(* IEC 61131-3 sources: NachHouse_CORE/V21/APP, 10 files *)

(* ---- _Nh_CFG.st ---- *)
VAR_GLOBAL
//	yVer	AT mRam[20000]	: NH_DBX_VER;            // verzia sa umiestni dalej do virtualne pamati. Na zaciatku sa pouzije a potom sa prepisuje datami
//   aDbx	AT mRam[0]	: NH_DBX;
   aCfg 	AT mRam[_Cfg0]	: ARRAY[1.._Nh_CFG] OF NH_CFG_CFG :=  [
			(cfg:='ROM',
                     ver:=1,
                     Siz   := SIZEOF(NH_ROM),                         // 1
                     al    := SIZEOF(NH_ROM.AL),
                     cx    := SIZEOF(NH_ROM.CX),
                     hw    := 0,                         // 1
                     io    := SIZEOF(NH_ROM.IO),                         // 1
                     me    := SIZEOF(NH_ROM.ME),                         // 1
                     cat   := 0,
                     fBr   := 14,
                     fSc   := 204,
                     mWsb  := 1,
                     mnu   := 25,
//                     wh    := 100,        // zobrazenie teploty v browse
                     ar2   := 1,
                     stp   := 0,

                     ref   := 252,
							del   := 1,
                     imp   := 1,
							bck	:= 1,
							RomIsZone:=1,

							NbrPoi:=1,
							),
         (cfg:='CAT',
                     ver:=0,
//                     Siz   := SIZEOF(NH_CAT),                         // 1
//                     al    := SIZEOF(NH_CAT.AL),
                     Siz   := 0,                         // 1
                     al    := 0,
                     cx    := 0,
                     hw    := 0,                         // 1
                     me    := 0,                         // 1
                     cat   := 0,
                     ar2   := 1,
                     stp   := 0,
                     fBr   := 12,
                     del   := 0,
                     ref   := 251,
							del   := 0,
                     imp   := 0,
							bck	:= 0,
                     ),

				(cfg:='ZON',
                     ver:=1,
                     Siz   := SIZEOF(NH_ROM),                         // 1
                     al    := SIZEOF(NH_ROM.AL),
                     cx    := SIZEOF(NH_ROM.CX),
                     hw    := 0,                         // 1
                     io    := SIZEOF(NH_ROM.IO),                         // 1
                     me    := SIZEOF(NH_ROM.ME),                         // 1
                     par   := 5,
                     fBr   := 14,
                     fSc   := 204,
                     mWsb  := 3,
                     mnu   := 24,
                     cat   := 0,
                     ar2   := 1,
                     stp   := 0,

                     ref   := 252,
							tgrp	:= 3,
							del   := 1,
                     imp   := 0,
							bck	:= 1,
							RomIsZone:=1,
			            ),
			(cfg:='SCN',                                                   // 4
                     ver:=1,
                     Siz   := SIZEOF(NH_SCN),
                     al    := SIZEOF(NH_SCN.AL),
                     cx    := SIZEOF(NH_SCN.CX),
                     me    := SIZEOF(NH_SCN.ME),
                     hw    := 0,                         // 1
							cat	:= 53,
                     sld   := 0,
                     par   := 10,
                     ou    := 1,
                     lst   := 1,
                     stp   := 1,
                     del   := 1,

                     fBr   := 5,
                     fSc   := 204,
                     mWsb  := 4,
                     mnu   := 93,
//                     analog:= 0,
                     tgrp  := 4,
//							analog:=true,
							zone	:=true,
							del   := 1,
                     imp   := 0,
							bck	:= 1,
							Visible:=1,
					      ),
			(cfg:='ACT',                                                   // 5
                     ver:=1,
                     Siz   := SIZEOF(NH_ACT),
                     al    := SIZEOF(NH_ACT.AL),
                     cx    := 0,
                     fBr   := 5,
                     fSc   := 204,
                     par   := 0,
                     cat   := 0,
							mWsb	:= 5,
                     mnu   := 94,
                     lst   := 1,
                     stp   := 1,
                     ou    := 0,
                     analog:= 0,
                     tgrp  := 5,
							zone	:=true,
							del   := 1,
                     imp   := 0,
							bck	:= 1,
							RomIsZone:=1,
							Visible:=1,
			            ),

         (cfg:='HET',                            		                    // 6
                     ver:=1,
                     Siz   := SIZEOF(NH_HET),
                     al    := SIZEOF(NH_HET.AL),
                     cx    := SIZEOF(NH_HET.CX),
                     hw    := 0,
                     me    := SIZEOF(NH_HET.ME),
                     io    := SIZEOF(NH_HET.IO),
                     fBR   := 23,
                     fSc   := 204,
                     mnu   := 28,
                     par   := 9,
          				mWsb	:= 6,
			            cat   := 5,
//                     cou   := 2,
                     sld   := 0,
//                     wh    := 100,        // zobrazenie teploty v browse
                     ou    := 0,       // ???? 23.11.2021
                     ref   := 251,
                     tgrp  := 6,
                    	lst	:= 1,
							del   := 1,
                     imp   := 0,
							bck	:= 1,
							ShwSta:=true,

							NbrPoi:=2,
							Imp_AL:=1,
                     ),

			(cfg:='KOT',                            	                       // 7
                     ver:=1,
                     Siz   := SIZEOF(NH_TVE),
                     al    := SIZEOF(NH_TVE.AL),
                     cx    := SIZEOF(NH_TVE.CX),
                     hw    := SIZEOF(NH_TVE.HW),
                     io    := SIZEOF(NH_TVE.IO),
                     me    := SIZEOF(NH_TVE.ME),
                     fBR   := 22,
                     mnu   := 36,
                     fSc   := 204,
                     cat   := 39,
                     sld   := 0,
                     par   := 0,
                     ou    := 1,
							del   := 0,
                     imp   := 1,
							bck	:= 1,
							Imp_AL:=1,
                     ),

			(cfg:='TVE',                            	                       // 8
                     ver:=1,
                     Siz   := SIZEOF(NH_TVE),
                     al    := SIZEOF(NH_TVE.AL),
                     cx    := SIZEOF(NH_TVE.CX),
                     hw    := SIZEOF(NH_TVE.HW),
                     io    := SIZEOF(NH_TVE.IO),
                     me    := SIZEOF(NH_TVE.ME),
                     fBR   := 22,
                     mnu   := 36,
                     fSc   := 204,
                     cat   := 39,
                     sld   := 0,
                     par   := 0,
                     ou    := 1,
							del   := 0,
                     imp   := 1,
							bck	:= 1,
							Imp_AL:=1,

                     ),
			(cfg:='CER',                               							  // 9
                     ver:=1,
                     Siz   := SIZEOF(NH_TVE),
                     al    := SIZEOF(NH_TVE.AL),
                     cx    := SIZEOF(NH_TVE.CX),
                     hw    := SIZEOF(NH_TVE.HW),
                     io    := SIZEOF(NH_TVE.IO),
                     me    := SIZEOF(NH_TVE.ME),
                     fBR   := 22,
                     mnu   := 36,
                     fSc   := 204,
                     cat   := 39,
                     sld   := 0,
                     par   := 0,
                     ou    := 1,
							del   := 0,
                     imp   := 1,
							bck	:= 1,
							Imp_AL:=1,

			            ),
         (cfg:='SVD',                                                      // 10
                     ver:=1,
                     Siz   := SIZEOF(NH_SVD),
                     al    := SIZEOF(NH_SVD.AL),
                     cx    := SIZEOF(NH_SVD.CX),
                     hw    := SIZEOF(NH_SVD.HW),
                     cat   := 1,
                     sld   := 0,
							lst	:= 1,
                     par   := 1,
                     ou    := 1,
                     fBr   := 43,
                     fSc   := 204,
                     mnu   := 45,
                     mWsb  := 10,
							ShwSta:=true,
                     del   := 0,
                     imp   := 1,
							bck	:= 1,
//                     adObr2:= 1,
			            ),
			(cfg:='SVA',                                                      // 11
                     ver:=1,
                     Siz   := SIZEOF(NH_SVA),
                     al    := SIZEOF(NH_SVA.AL),
                     cx    := SIZEOF(NH_SVA.CX),
                     hw    := SIZEOF(NH_SVA.HW),
                     cat   := 1,
							lst	:= 1,
                     sld   := 1,
                     par   := 2,
                     ou    := 1,
                     fBr   := 43,
                     fSc   := 204,
                     mWsb  := 11,
                     mnu   := 45,
                     analog:=true,
							ShwSta:=true,
                     del   := 0,
                     imp   := 1,
							bck	:= 1,
			            ),
			(cfg:='RGB',                                                      // 12
                     ver:=1,
                     Siz   := SIZEOF(NH_RGB),
                     al    := SIZEOF(NH_RGB.AL),
                     cx    := SIZEOF(NH_RGB.CX),
                     hw    := SIZEOF(NH_RGB.HW),
                     cat   := 1,
                     sld   := 1,
							lst	:= 1,
                     par   := 3,
                     ou    := 1,
                     fBr   := 43,
                     fSc   := 204,
                     mWsb  := 11,
                     mnu   := 46,
                     analog:=true,
                     del   := 0,
                     imp   := 1,
							bck	:= 1,
                     ),
			(cfg:='WSB',                                                      // 13
                     ver:=1,
                     Siz   := SIZEOF(NH_WSB),
                     al    := SIZEOF(NH_WSB.AL),
                     cx    := SIZEOF(NH_WSB.CX),
                     hw    := SIZEOF(NH_WSB.HW),
                     me    := SIZEOF(NH_WSB.ME),
                     fSc   := 204,
                     mnu   := 27,
                     cat   := 24,
                     sld   := 0,
                     par   := 4,
                     ref   := 252,
                     body  := 1,
                     tgrp  := 13,
                     del   := 0,
                     imp   := 1,
							bck	:= 1,
							led	:= 1,
                     ),
			(cfg:='TLA',                                       			     // 14

                     ver:=1,
                     Siz   := SIZEOF(NH_TLA),
                     al    := SIZEOF(NH_TLA.AL),
                     cx    := SIZEOF(NH_TLA.CX),
                     hw    := SIZEOF(NH_TLA.HW),
                     me    := SIZEOF(NH_TLA.ME),
                     fSc   := 204,
                     mnu   := 27,

//                     iov   := 1,
                     cat   := 24,
                     sld   := 0,
                     par   := 4,
                     ref   := 252,
                     body  := 1,
                     tgrp  := 13,
                     del   := 0,
                     imp   := 1,
							bck	:= 1,
                     ),
   	   (cfg:='PIR',                                                     // 15
                     ver:=1,
                     Siz   := SIZEOF(NH_PIR),
                     al    := SIZEOF(NH_PIR.AL),
                     cx    := SIZEOF(NH_PIR.CX),
                     hw    := SIZEOF(NH_PIR.HW),
                     me    := 0,	//SIZEOF(NH_PIR.ME),
                     cat   := 15,
                     fBr   := 15,
                     fSc   := 204,
                     mWsb  := 15,
                     mnu   := 56,
                     par   := 7,
                     body  := 1,
                     tgrp  := 15,
                     del   := 0,
                     imp   := 1,
							bck	:= 1,
                     ),

			(cfg:='TER',                                                      // 16
                     ver:=1,
                     Siz   := SIZEOF(NH_TER),
                     al    := SIZEOF(NH_TER.AL),
                     cx    := SIZEOF(NH_TER.CX),
                     hw    := SIZEOF(NH_TER.HW),
                     me    := SIZEOF(NH_TER.ME),
                     cat   := 14,
//                     wh    := 100,        // zobrazenie teploty v browse
                     par   := 0,
                     fBr   := 20,
                     fSc   := 204,
                     mnu   := 34,
                     tgrp  := 16,
							//   iov	:= 100,
							ShwSta:=false,
							analog:=true,
							zone	:=true,
                     del   := 1,
                     imp   := 1,
							bck	:= 1,
                     ),

			(cfg:='TEH',                                                      // 17
                     ver:=1,
                     Siz   := SIZEOF(NH_TER),
                     al    := SIZEOF(NH_TER.AL),
                     cx    := SIZEOF(NH_TER.CX),
                     hw    := SIZEOF(NH_TER.HW),
                     me    := SIZEOF(NH_TER.ME),
//                     wh    := 100,        // zobrazenie teploty v browse
                     cat   := 39,
                     par   := 0,
                     fBr   := 20,
                     fSc   := 204,
                     mnu   := 34,
                     tgrp  := 16,
                     //iov   := 100,
							analog:=true,
                     del   := 1,
                     imp   := 1,
							bck	:= 1,
                     ),
			(cfg:='TEK',                                                      // 18
                     ver:=1,
                     Siz   := SIZEOF(NH_TER),
                     al    := SIZEOF(NH_TER.AL),
                     cx    := SIZEOF(NH_TER.CX),
                     hw    := SIZEOF(NH_TER.HW),
                     me    := SIZEOF(NH_TER.ME),
//                     wh    := 100,        // zobrazenie teploty v browse
                     cat   := 39,
                     par   := 0,
                     fBr   := 20,
                     fSc   := 204,
                     mnu   := 34,
							analog:=true,
                     tgrp  := 16,
                     //  iov   := 100,
                     del   := 1,
                     imp   := 1,
							bck	:= 1,
                     ),
			(cfg:='LUX',                                                      // 19
                     ver:=1,
                     Siz   := SIZEOF(NH_LUX),
                     al    := SIZEOF(NH_LUX.AL),
                     cx    := SIZEOF(NH_LUX.CX),
                     hw    := SIZEOF(NH_LUX.HW),
                     me    := SIZEOF(NH_LUX.ME),
//                     wh    := 101,        // zobrazenie % v browse
                     cat   := 16,
                     par   := 0,
                     fBr   := 20,

                     fSc   := 204,
                     mnu   := 59,

                     tgrp  := 16,
                     //  iov   := 101,
							analog:=true,
							zone	:=true,
                     del   := 0,
                     imp   := 1,
							bck	:= 1,
                     ),
                                                                           // 20
	      (cfg:='FAV',
                     ver:=1,
                     Siz   := SIZEOF(NH_FAV),
                     al    := 0,
                     cx    := SIZEOF(NH_FAV.CX),
                     fav   := 0,
                     par   := 0,

                     del   := 1,
                     imp   := 0,
							bck	:= 0,
                     ),

	      (cfg:='ZAS',                                                        // 21
                     ver:=1,
                     Siz   := SIZEOF(NH_SVD),
                     al    := SIZEOF(NH_SVD.AL),
                     cx    := SIZEOF(NH_SVD.CX),
                     hw    := SIZEOF(NH_SVD.HW),
                     cat   := 2,
							lst	:= 1,
                     par   := 1,
                     sld   := 0,
                     ou    := 1,
                     fBr   := 43,
                     fSc   := 204,
                     mnu   := 45,
                     mWsb  := 10,
                     del   := 0,
                     imp   := 1,
							bck	:= 1,

//                     adObr2:= 1,
                     ),

			(cfg:='USR',
                     ver:=1,
                     Siz   := SIZEOF(NH_USR),  					              // 22  uzivatelia
                     al    := 0,
                     cx    := SIZEOF(NH_USR.CX),
                     stp   := 0,
                     cat   := 31,
                     par   := 0,
                     ref   := 254,

                     del   := 1,
                     imp   := 0,
							bck	:= 1,
                     ),
			(cfg:='VEN',                                                      // 23 TVE pre Vetranie // ako TVE pre HET
                     ver:=1,
                     Siz   := SIZEOF(NH_TVE),
                     al    := SIZEOF(NH_TVE.AL),
                     cx    := SIZEOF(NH_TVE.CX),
                     hw    := SIZEOF(NH_TVE.HW),
                     io    := SIZEOF(NH_TVE.IO),
                     me    := SIZEOF(NH_TVE.ME),
//							tgr	:= 101,
							//   //  iov	:= 101,
                     fBR   := 22,
                     mnu   := 36,
                     fSc   := 204,
                     cat   := 4,      // globalne nastavenaia/vetranie
                     sld   := 1,
                     par   := 0,
                     ou    := 1,
                     del   := 0,
                     imp   := 1,
							bck	:= 1,
							Imp_AL:=1,

                     ),
			(cfg:='KEY',                                                      // 24  klavesnice
                     ver:=1,
                     Siz   := SIZEOF(NH_KEY),
                     al    := SIZEOF(NH_KEY.AL),
                     cx    := SIZEOF(NH_KEY.CX),
                     hw    := SIZEOF(NH_KEY.HW),
                     me    := SIZEOF(NH_KEY.ME),
                     cat   := 25,
                     body  := 1,
                     tgrp  := 24,
                     del   := 0,
                     imp   := 1,
							bck	:= 1,
                     ),

         (cfg:='GLB',
                     ver:=1,
                     Siz   := SIZEOF(NH_GLB), 				               // 25 Globana konfiguracia
                     al    := 0,
                     cx    := SIZEOF(NH_GLB.CX),
                     al    := 0,
                     cf    := 0,
                     hw    := 0,
                     me    := 0,

                     ImpFullCfg:=1,
                     ImpFullRec:=1,             // nema klasicke CFG_ALL obnovi naraz cele cfg[].siz
                     del   := 0,
                     imp   := 0,
							bck	:= 0,
                     ),
         (cfg:='POI',
                     ver:=2,
                     Siz   := SIZEOF(NH_POI), 				               // 26   zoznam casovych pointov
                     al    := 0,
                     cx    := SIZEOF(NH_POI.CX),
                     al    := 0,
                     cf    := 0,
                     hw    := 0,
                     me    := 0,

                     ImpFullCfg:=1,
                     ImpFullRec:=1,
                     del   := 0,
                     imp   := 0,
							bck	:= 0,
                     ),
			(cfg:='H2O',                                                   // 27
                     Siz   := SIZEOF(NH_DOR),
                     al    := SIZEOF(NH_DOR.AL),
                     cx    := SIZEOF(NH_DOR.CX),
                     hw    := SIZEOF(NH_DOR.HW),
							me		:= 0,
                     cat   :=47,
                     tgrp  :=16,
                     del   := 0,
                     imp   := 1,
							bck	:= 1,
                     ),
			(cfg:='FIR',                                                   // 28
                     Siz   := SIZEOF(NH_DOR),
                     al    := SIZEOF(NH_DOR.AL),
                     cx    := SIZEOF(NH_DOR.CX),
                     hw    := SIZEOF(NH_DOR.HW),
							me		:= 0,
                     cat   :=46,
                     tgrp  :=16,
                     del   := 0,
                     imp   := 1,
							bck	:= 1,
                     ),
			(cfg:='GAS',                                                   // 29
                     ver:=1,
                     Siz   := SIZEOF(NH_DOR),
                     al    := SIZEOF(NH_DOR.AL),
                     cx    := SIZEOF(NH_DOR.CX),
                     hw    := SIZEOF(NH_DOR.HW),
							me		:= 0,
                     cat   := 50,
                     tgrp  :=16,
                     del   := 0,
                     imp   := 1,
							bck	:= 1,
                     ),
         (cfg:='MAR',                                                   // 30 horizontalne tienenie (markiza,pergola)
                     ver:=1 ,
                     Siz   := SIZEOF(NH_ROL),
                     al    := SIZEOF(NH_ROL.AL),
                     cx    := SIZEOF(NH_ROL.CX),
                     hw    := SIZEOF(NH_ROL.HW),
                     me    := SIZEOF(NH_ROL.ME),
                     par   := 11,
                     cat   := 3,
                     tgrp  :=31,
                     sld   := 0,
                     ou    := 1,
                     del   := 0,
                     imp   := 1,
							bck	:= 1,
                     ),
 	      (cfg:='ROL',                                                    // 31 rolety = vertikalne tienenie
                     ver:=1,
                     Siz   := SIZEOF(NH_ROL),
                     al    := SIZEOF(NH_ROL.AL),
                     cx    := SIZEOF(NH_ROL.CX),
                     hw    := SIZEOF(NH_ROL.HW),
                     me    := SIZEOF(NH_ROL.ME),
                     par   := 12,
                     cat   := 3,
                     tgrp  :=31,
                     fBr   := 8,
                     fSc   := 204,
                     mnu   := 63,
                     mWsb  := 31,
                     sld   := 1,
                     ref   := 252,
                     del   := 0,
                     imp   := 1,
							bck	:= 1,
                     ),
 	      (cfg:='SIR',                                                      // 32
                     ver:=1,
                     Siz   := SIZEOF(NH_SVD),
                     al    := SIZEOF(NH_SVD.AL),
                     cx    := SIZEOF(NH_SVD.CX),
                     hw    := SIZEOF(NH_SVD.HW),
                     cat   := 6,
                     sld   := 0,
							lst	:= 1,
                     par   := 1,
                     ou    := 1,
                     fBr   := 43,
                     fSc   := 204,
                     mnu   := 45,
                     del   := 0,
                     imp   := 1,
							bck	:= 1,
                     ),
			(cfg:='DOR',                             									// 33
                     ver:=1,
                     Siz   := SIZEOF(NH_DOR),
                     al    := SIZEOF(NH_DOR.AL),
                     cx    := SIZEOF(NH_DOR.CX),
                     hw    := SIZEOF(NH_DOR.HW),
							me		:= 0,
                     cat   := 45,
                     par   := 0,
							fbr	:= 15,
                     fSc   := 204,
                     mnu   := 56,
                     body  := 1,
                     tgrp  :=16,
							//   //  iov	:=33,
                     del   := 0,
                     imp   := 1,
							bck	:= 1,
							lst	:= 1,
                     ),
			(cfg:='WIN',                     									      // 34
                     Siz   := SIZEOF(NH_DOR),
                     al    := SIZEOF(NH_DOR.AL),
                     cx    := SIZEOF(NH_DOR.CX),
                     hw    := SIZEOF(NH_DOR.HW),
							me		:= 0,
                     cat   := 44,
                     par   := 0,
                     body  := 1,
                     tgrp  :=16,
							//   //  iov	:= 0,
                     del   := 0,
                     imp   := 1,
							bck	:= 1,
							lst	:= 1,
                     ),
 	      (cfg:='BLK',                                                       // 35 BLIKAC VSEOBECNY
                     ver:=1,
                     Siz   := SIZEOF(NH_BLK),
                     al    := SIZEOF(NH_BLK.AL),
                     cx    := SIZEOF(NH_BLK.CX),
							hw		:= 0,
							io		:= 0,
                     me    := SIZEOF(NH_BLK.ME),
                     fBr   := 19,
                     fSc   := 204,
                     mnu   := 41,
                     lst   := 1,
                     stp   := 1,
                     del   := 1,
							zone	:=true,
                     NoRecCat := 1,
                     del   := 1,
                     imp   := 0,
							bck	:= 1,
							RomIsZone:=1,
							Visible:=1,
                     ),

 	      (cfg:='BLX',                                                       // 36 blikac len pre DEV
                     ver:=1,
                     Siz   := SIZEOF(NH_BLK),
							cf		:= 0,
                     al    := 0,
                     cx    := SIZEOF(NH_BLK.CX),
							hw		:= 0,
							io		:= 0,
                     me    := SIZEOF(NH_BLK.ME),

                     NoRecCat := 1,
                     del   := 0,
                     imp   := 0,
							bck	:= 0,
                     ),

         (cfg:='GAT',                                                   // 37 garaz,brana,branicka,zavora
                     ver:=1,
                     Siz   := SIZEOF(NH_GAT),
                     al    := SIZEOF(NH_GAT.AL),
                     cx    := SIZEOF(NH_GAT.CX),
                     hw    := SIZEOF(NH_GAT.HW),
							io		:= SIZEOF(NH_GAT.IO),
							me		:= SIZEOF(NH_GAT.ME),
							mWsb	:= 37,
                     fBr   := 48,
                     fSc   := 204,
                     mnu   := 53,
                     par   := 13,
							lst	:= 1,
                     cat   := 7,
                     stp   := 1,
                     sld   := 1,
                     ou    := 1,
                     del   := 0,
                     imp   := 1,
							bck	:= 1,
                     ),

         (cfg:='RFI',                                                   // 38 RFI snimace
                     Siz   := SIZEOF(NH_RFI),
                     al    := SIZEOF(NH_RFI.AL),
                     cx    := SIZEOF(NH_RFI.CX),
                     hw    := SIZEOF(NH_RFI.HW),
                     cat   := 27,
                     par   := 0,
                     del   := 0,
                     imp   := 1,
							bck	:= 1,
                     ),
         (cfg:='RFK',                                                   // 39 RFK - karty
                     Siz   := SIZEOF(NH_RFK),
                     al    := 0,
                     cx    := SIZEOF(NH_RFK.CX),
                     cat   := 37,
                     par   := 0,

                     del   := 0,
                     imp   := 0,
							bck	:= 1,
                     ),
			(cfg:='TGL',                                                     // 40 TOuch Glass
                     ver:=1,
                     Siz   := SIZEOF(NH_TGL),
                     al    := SIZEOF(NH_TGL.AL),
                     cx    := SIZEOF(NH_TGL.CX),
                     hw    := SIZEOF(NH_TGL.HW),
                     me    := SIZEOF(NH_TGL.ME),
                     fSc   := 204,
                     mnu   := 27,
//                     //  iov   := 1,
                     cat   := 24,
                     sld   := 0,
                     par   := 15,
//                     wsb   := 1,
                     ref   := 252,
                     body  := 1,
                     tgrp  :=13,
                     del   := 1,
                     imp   := 1,
							bck	:= 1,
							led	:= 1,
							dis	:= 1,
                     ),
			(cfg:='COX',                                     // 41  - nanalogove snimanie CO2,CO,BUT
                     ver:=1,
                     Siz   := SIZEOF(NH_LUX),
                     al    := SIZEOF(NH_LUX.AL),
                     cx    := SIZEOF(NH_LUX.CX),
                     hw    := SIZEOF(NH_LUX.HW),
                     me    := SIZEOF(NH_LUX.ME),
//                     wh    := 101,        // zobrazenie % v browse
                     cat   := 48,
                     par   := 0,
                     fBr   := 20,
                     fSc   := 204,
                     mnu   := 59,
                     tgrp  := 0,
                     //  iov   := 101,
							analog:=true,
							zone	:=true,
                     del   := 0,
                     imp   := 1,
							bck	:= 1,
                     ),
         (cfg:='DLM',                            		     // 42        DALI-MASTER 62
                     ver:=1,
                     Siz   := SIZEOF(NH_DLM),
                     al    := SIZEOF(NH_DLM.AL),
                     cx    := SIZEOF(NH_DLM.CX),
                     me    := SIZEOF(NH_DLM.ME),                          // vsetko je v HW
                     hw    := SIZEOF(NH_DLM.HW),
							mWsb	:= 4,
                     cat   := 35,
                     sld   := 1,
                     par   := 16,
                     ar2   := 0,
                     stp   := 0,
                     fBr   := 3,
                     fSc   := 204,
                     mnu   := 4,
                     ou    := 1,
//                     adObr2:= 1,

                     lvl254   := 1,
                     analog:=true,
                     dali     := 1,
                     del   := 0,
                     imp   := 1,
							bck	:= 1,
                     ),
         (cfg:='DLS',                            		     // 43        DALI-slave
                     ver:=1,
                     Siz   := SIZEOF(NH_DLS),
                     al    := SIZEOF(NH_DLS.AL),
                     cx    := SIZEOF(NH_DLS.CX),
                     me    := SIZEOF(NH_DLS.ME),
                     hw    := 0,                         // ma uplne inu srokturu, tak je 0  NH_DLS_HW
							mWsb	:=11,
                     cat   := 1,
                     sld   := 1,                            // slider sa nadefinuje sa az
//                     lst   := 1,
                     lst   := 0,
                     par   := 16,
                     ar2   := 0,
                     stp   := 1,
                     fBR   := 5,
                     fSc   := 204,
                     mnu   := 4,             // user menu - len parametre
                     ou    := 1,
//                     adObr2:= 1,

                     imp   := 0,
                     lvl254   := 1,
                     analog:=true,
                     dali     := 1,
                     del   := 0,
                     imp   := 0,
							bck	:= 1,
                     ),
         (cfg:='DLG',                            		     // 44        DALI-Group
                     ver:=1,
                     Siz   := SIZEOF(NH_DLG),
                     al    := SIZEOF(NH_DLG.AL),                     hw    := 0,                         // ma uplne inu srokturu, tak je 0  NH_DLS_HW
                     cx    := SIZEOF(NH_DLG.CX),
                     me    := SIZEOF(NH_DLG.ME),
							mWsb	:= 4,
                     cat   := 54,
                     sld   := 1,
                     lst   := 1,
                     //scn   := 1,
                     ar2   := 0,
                     stp   := 1,
                     fBr   := 5,
                     fSc   := 204,
                     mnu   := 4,
                     par   := 16,
                     ou    := 1,
//                     adObr2:= 1,

                     imp   := 0,
                     lvl254   := 1,
                     analog:=true,
                     dali     := 1,
                     del   := 0,
                     imp   := 0,
							bck	:= 1,
							Visible:=1,
                     ),
	      (cfg:='SMW',                                                        // 45    Smart WAY
                     ver:=1,
                     Siz   := SIZEOF(NH_SMW),
                     al    := SIZEOF(NH_SMW.AL),
                     cx    := 0,
                     cat   := 0,
                     par   := 0,
                     sld   := 0,

                     NoRecCat := 1,
                     del   := 0,
                     imp   := 0,
							bck	:= 0,

                     ),

 	      (cfg:='MSG',                                                       // 46 SPRAVY
                     ver:=1,
                     Siz   := SIZEOF(NH_MSG),
                     al    := SIZEOF(NH_MSG.AL),
//                     cx    := SIZEOF(NH_MSG.CX),
                     me    := 0, 	// SIZEOF(NH_BLK.ME),
                     fBr   := 19,
//                     fSc   := 204,
//                     mna   := 41,
//                     mnu   := 41,
//                     lst   := 1,
                     stp   := 1,
                     del   := 1,

//                     NoRecCat := 1,
                     del   := 0,
                     imp   := 0,
							bck	:= 1,
                     RomIsZone:=1,
                     ),
         (cfg:='HEV',                            		                    // 47 - regulator vetrania
                     ver:=1,
                     Siz   := SIZEOF(NH_HET),
                     al    := SIZEOF(NH_HET.AL),
                     cx    := SIZEOF(NH_HET.CX),
                     hw    := 0,
                     me    := SIZEOF(NH_HET.ME),
                     io    := SIZEOF(NH_HET.IO),
                     fBR   := 23,
                     fSc   := 204,
                     mnu   := 28,
                     par   := 9,
							mWsb	:= 6,
                     cat   := 4,
//                     cou   := 2,
                     sld   := 0,
//                     wh    := 100,        // zobrazenie teploty v browse
                     ou    := 0,       // ???? 23.11.2021
                     ref   := 251,
                     tgrp  := 6,
                    	lst	:= 1,
                     del   := 1,
                     imp   := 0,
							bck	:= 1,
							ShwSta:=true,

							NbrPoi:=2,
							Imp_AL:=1,
                     ),
			(cfg:='ALA',                                                   // 48 - akcie zabezpecovacky
                     ver:=1,
                     Siz   := SIZEOF(NH_ALA),
                     al    := SIZEOF(NH_ALA.AL),
                     cx    := SIZEOF(NH_ALA.CX),
//                     me    := SIZEOF(NH_ACA.ME),
                     fBr   := 19,
                     fSc   := 90,
                     mnu   := 49,
                     par   :=  0,
                     cat   := 55,
                     lst   := 1,
                     stp   := 1,
                     ou    := 0,
                     tgrp  := 5,

							del   := 1,
                     imp   := 0,
							bck	:= 1,
				         RomIsZone:=1,
						   ),

			(cfg:='VVO',                                                   // 49 - ventil vody
                     ver:=1,
                     Siz   := SIZEOF(NH_VVO),
                     al    := SIZEOF(NH_VVO.AL),
                     cx    := SIZEOF(NH_VVO.CX),
                     hw    := SIZEOF(NH_VVO.HW),
                     cat   := 6,
                     sld   := 0,
							lst	:= 1,
                     par   := 1,
                     ou    := 1,
                     fBr   := 43,
                     fSc   := 204,
                     mnu   := 87,
							ShwSta:=true,
                     del   := 1,
                     imp   := 1,
							bck	:= 1,
						   ),

			(cfg:='TIM',                                                   // 50 - akcie zabezpecovacky
                     ver:=1,
                     Siz   := SIZEOF(NH_TIM),
                     al    := SIZEOF(NH_TIM.AL),
                     cx    := SIZEOF(NH_TIM.CX),
                     me    := SIZEOF(NH_TIM.ME),
                     fBr   := 15,
                     fSc   := 204,
                     mnu   := 71,

                     lst   := 0,
                     stp   := 1,
                     del   := 1,
							zone	:= 1,
                     NoRecCat := 1,
                     imp   := 0,
							bck	:= 1,
							RomIsZone:=1,
							Visible:=1,
						   ),
			(cfg:='RHX',                                     					// 51  - vlhkost - RH
                     ver:=1,
                     Siz   := SIZEOF(NH_LUX),
                     al    := SIZEOF(NH_LUX.AL),
                     cx    := SIZEOF(NH_LUX.CX),
                     hw    := SIZEOF(NH_LUX.HW),
                     me    := SIZEOF(NH_LUX.ME),
//                     wh    := 101,        // zobrazenie % v browse
                     cat   := 17,
                     par   := 0,
                     fBr   := 20,
                     fSc   := 204,
                     mnu   := 59,
                     tgrp  := 0,
                     //  iov   := 101,
							analog:=true,
							zone	:=true,
                     del   := 0,
                     imp   := 1,
							bck	:= 1,
                     )

 	];

         eROM  {HIDDEN} :  NH_ROM;
//			eCAT  {HIDDEN} :  NH_OK;
			eZON  {HIDDEN} :  NH_ROM;
			eSCN  {HIDDEN} :  NH_SCN;
	      eACT  {HIDDEN} :  NH_ACT;
			eHET  {HIDDEN} :  NH_HET :=
					(cf := (cat := 5));
			eKOT  {HIDDEN} :  NH_TVE :=
					(cf := (cat := 5),
					 cx := (
 						 reg:= (	ModeFromSrc := 0,
						 			Guard 		:= 1,
 									Mode 			:= 0,
						 			Delay 		:= 0,
						 			reg := [( Wht := 0,
									 				out := [   0,   25,   50,  100],
									 				req := [ 5.0, 22.0, 26.0, 29.0]
									 			),
											  ( Wht := 0,
											  		out := [   0,   25,   50, 100],
											  		req := [ 0.0, 25.0, 22.0, 19.0]
									 		    )
												]),
									guard := (	tDis:=22,
													val := [20,40,21,27],
												 ),
									),
 					);
			eTVE  {HIDDEN} :  NH_TVE :=
					(cf := (cat := 5),
					 cx := (
 						 reg:= (	ModeFromSrc := 1,
						 			Guard 		:= 1,
 									Mode 			:= 0,
						 			Delay 		:= 0,
						 			reg := [( Wht := 0,
									 				out := [   0,  100,  100,  100],
									 				req := [ 5.0, 22.0, 26.0, 29.0]
									 			),
											  ( Wht := 0,
											  		out := [   0,  100,  100,  100],
											  		req := [ 0.0, 25.0, 22.0, 20.0]
									 		    )
												]),
									guard := (	tDis:=17,
													val := [5,30,21,27],
												 ),
									),
 					);
			eCER  {HIDDEN} :  NH_TVE:=     // 9  CER
					(cf := (cat := 5),
					 cx := (
 						 reg:= (	ModeFromSrc := 1,
						 			Guard 		:= 0,
 									Mode 			:= 0,
						 			Delay 		:= 0,
						 			reg := [( Wht := 0,
									 				out := [   0,  100,  100,  100],
									 				req := [ 5.0, 22.0, 26.0, 29.0]
									 			),
											  ( Wht := 0,
											  		out := [   0,  100,  100,  100],
											  		req := [ 0.0, 25.0, 22.0, 20.0]
									 		    )
												]),
									guard := (	tDis:=17,
													val := [5,30,21,27],
												 ),
									),
 					);
         eSVD  {HIDDEN} :  NH_SVD;    // 10
			eSVA  {HIDDEN} :  NH_SVA;
			eRGB  {HIDDEN} :  NH_RGB;
			eWSB  {HIDDEN} :  NH_WSB;
			eTLA  {HIDDEN} :  NH_TLA;
   	   ePIR  {HIDDEN} :  NH_PIR;    // 15
			eTER  {HIDDEN} :  NH_TER;
			eTEH  {HIDDEN} :  NH_TER;
			eTEK  {HIDDEN} :  NH_TER;
			eLUX  {HIDDEN} :  NH_LUX;
	      eFAV  {HIDDEN} :  NH_FAV;    // 20
	      eZAS  {HIDDEN} :  NH_SVD;
			eUSR  {HIDDEN} :  NH_USR;
			eVEN  {HIDDEN} :  NH_TVE :=
					(cf := (cat := 4),
					 cx := (
 						 reg:= (
						  			ModeFromSrc := 0,
						 			Guard 		:= 0,
 									Mode 			:= 0,
						 			Delay 		:= 0,
						 			reg := [( Wht := 0,
									 				out := [   0,  100,  100,  100],
									 				req := [ 0.0, 25.0, 33.0, 40.0]
									 			),
											  ( Wht := 1,
											  		out := [   0,  100,  100,  100],
											  		req := [ 0.0, 24.0, 22.5, 21.0]
									 		    )
												]),
									),
 					);
			eKEY  {HIDDEN} :  NH_KEY;
	      eGLB  {HIDDEN} :  NH_GLB;     // 25
	      ePOI  {HIDDEN} :  NH_POI;     // 26
			eH2O  {HIDDEN} :  NH_DOR;
			eFIR  {HIDDEN} :  NH_DOR;
			eGAS  {HIDDEN} :  NH_DOR;
         eMAR  {HIDDEN} :  NH_ROL;     // 30
 	      eROL  {HIDDEN} :  NH_ROL;     // 31
 	      eSIR  {HIDDEN} :  NH_SVD;
			eDOR  {HIDDEN} :  NH_DOR;     // 33
			eWIN  {HIDDEN} :  NH_DOR;
 	      eBLK  {HIDDEN} :  NH_BLK;      // 35
 	      eBLX  {HIDDEN} :  NH_BLK;
 	      eGAT  {HIDDEN} :  NH_GAT;      // 37
 	      eRFI  {HIDDEN} :  NH_RFI;
 	      eRFK  {HIDDEN} :  NH_RFK;
 	      eTGL  {HIDDEN} :  NH_TGL;      // 40
			eCOX  {HIDDEN} :  NH_LUX;      // 41: RH,CO2,CO
			eDLM  {HIDDEN} :  NH_DLM;      // 42: Dali Master
			eDLS  {HIDDEN} :  NH_DLS;      // 43: Dali Slave
			eDLG  {HIDDEN} :  NH_DLG;      // 44: Dali Slave
	      eSMW  {HIDDEN} :  NH_SMW;      // 45: presunute z aCfg[25]
	      eMSG  {HIDDEN} :  NH_MSG;      // 46: SMS/MAIL/MSG
			eHEV  {HIDDEN} :  NH_HET	:=        // 47  regulator vetrania
					(cf := (cat := 4),
					 cx := (
 						 reg:= (
						  			ModeFromSrc := 1,
						 			Guard 		:= 0,
 									Mode 			:= 0,
						 			Delay 		:= 0,

						 			reg := [( Wht := 1,
									 				out := [   0,   25,   50,  100],
									 				req := [ 0.0, 70.0, 50.0, 30.0],
													hys := [  2.0,  4.0,  6.0, 			// Dn
							 									 2.0,  4.0,  6.0],  	      // Up
									 			),
											  ( Wht := 1,
											  		out := [   0,   25,   50,  100],
											  		req := [ 0.0, 70.0, 50.0, 40.0],
													hys := [  2.0,  4.0,  6.0, 			// Dn
							 									 2.0,  4.0,  6.0],  	      // Up

									 		    )
												]

												),

									),
 					);

(*
				( cx := ( reg := (Mode := 0, ModeFromSrc := false,
							btn := [1,1,1,1,1,0],
							reg :=
						[( wht := 0,  pv := [( val := [ 0.0, 25.0, 50.0,100.0]),
													( val := [ 0.0, 70.0, 50.0, 30.0])]),
						 ( wht := 0,  pv := [( val := [ 5.0, 25.0, 50.0,100.0]),
													( val := [ 0.0, 70.0, 50.0, 40.0])])]),
				));
*)
			eALA  {HIDDEN} :  NH_ALA := (ok:=(ok:=0));      // 48  akcie ALA
			eVVO  {HIDDEN} :  NH_VVO;		// 49 ventil vody
			eTIM  {HIDDEN} :  NH_TIM;		// 50 timer + rnd + sunset
			eRHX  {HIDDEN} :  NH_LUX;     // 51: RH - vlhkost

//			eRVE  {HIDDEN} :  NH_RVE;      // 45: regulator ventilatora/rekuperacie

	aPar	{HIDDEN}	AT mRam[ _Par0 ]	: ARRAY[1.._Nh_PAR] OF NH_PAR_CFG := [
			(cfg:='SVD',Siz:=SIZEOF(NH_SVD_PAR)),	         // 1
			(cfg:='SVA',Siz:=SIZEOF(NH_SVA_PAR)),	         // 2
			(cfg:='RGB',Siz:=SIZEOF(NH_RGB_PAR)),	         // 3
			(cfg:='WSB',Siz:=SIZEOF(NH_WSB_PAR)), 	         // 4
			(cfg:='ZON',Siz:=SIZEOF(NH_ZON_PAR)),    			// 5  ZON -> ACT
			(cfg:='XX1',Siz:=SIZEOF(NH_SVD_PAR)),	         // 6
			(cfg:='PIR',Siz:=SIZEOF(NH_PIR_PAR)), 	         // 7
			(cfg:='XX2',Siz:=SIZEOF(NH_SVD_PAR)),	         // 8
			(cfg:='HET',Siz:=SIZEOF(NH_HET_PAR)),           // 9
			(cfg:='SCN',Siz:=SIZEOF(NH_SVA_PAR),grp:=1),   // 10   SCN vo vazbe in, parameter sa prebera z hlavicky (DEV-LIST k SCN)
			(cfg:='MAR',Siz:=SIZEOF(NH_ROL_PAR)),          // 11   MAR - zatial pre markizy,este nepouzite
			(cfg:='ROL',Siz:=SIZEOF(NH_ROL_PAR),ver:=1),   // 12   ROL
			(cfg:='GAT',Siz:=SIZEOF(NH_GAT_PAR)),          // 13   BRA (garaz,brana,branicka)
			(cfg:='XX3',Siz:=SIZEOF(NH_SVD_PAR)),          // 14          VOLNY = byvaly ZON (PSN prikazy)
			(cfg:='TGL',Siz:=SIZEOF(NH_WSB_PAR)),          // 15   TGL
			(cfg:='DLS',Siz:=SIZEOF(NH_RGB_PAR))           // 16   DLS,DLG,DLM
	        ];

         epSVD  {HIDDEN} :  NH_SVD_PAR;	// 1
         epSVA  {HIDDEN} :  NH_SVA_PAR;   // 2
         epRGB  {HIDDEN} :  NH_RGB_PAR;   // 3
         epWSB  {HIDDEN} :  NH_WSB_PAR;   // 4
         epZON  {HIDDEN} :  NH_ZON_PAR;   // 5
         epXX1  {HIDDEN} :  NH_SVD_PAR;   // 6
         epPIR  {HIDDEN} :  NH_PIR_PAR;   // 7
         epXX2  {HIDDEN} :  NH_SVD_PAR;   // 8
         epHET  {HIDDEN} :  NH_HET_PAR;   // 9
         epSCN  {HIDDEN} :  NH_SVA_PAR;   // 10
         epMAR  {HIDDEN} :  NH_ROL_PAR;   // 11
         epROL  {HIDDEN} :  NH_ROL_PAR ;   // 12
         epGAT  {HIDDEN} :  NH_GAT_PAR;   // 13
         epXX3  {HIDDEN} :  NH_SVD_PAR;   // 14
         epTGL  {HIDDEN} :  NH_WSB_PAR;   // 15
         epDLS  {HIDDEN} :  NH_RGB_PAR := ( all := ( lvl := 100), rgb := ( lvl := [254,254,254,254,254]));  // 16

//	aVaz	{HIDDEN}	AT mRam[ _Vaz0 ]	: ARRAY[1.._Nh_VAZ] OF NH_VAZ_CFG ;

	aVaz	{HIDDEN}	AT mRam[ _Vaz0 ]	: ARRAY[1.._Nh_VAZ] OF NH_VAZ_CFG := [
			(cfg:='VZ1'),
			(cfg:='VZ2'),
			(cfg:='VZ3'),
			(cfg:='VZ4'),
			(cfg:='VZ5',siz:=0),
			(cfg:='VZ6',siz:=0),
			(cfg:='VZ7',siz:=0),
			(cfg:='VZ8',siz:=0),
			(cfg:='VZ9',siz:=0) ];

         eVAZ  :  NH_VAZ;     // 33

(* aVaz[1]  :  HOME page (dash+qick) menu
               in.c = usr (0=default), in.n := -1 dash, -2 quick, -3...
   aVaz[2]  :  FAV
               in.c = usr (0=vsetci), in.n := cislo FAV 0=vsetci dash, -2 quick, -3...

*)
(*
	aWrk	: ARRAY[1.._Nh_WRK] OF NH_WRK := [
			(Siz := SIZEOF(NH_ROM_WRK), cfg := 1),	                // 1 = Rom
			(Siz := SIZEOF(NH_CAT_WRK), cfg := 2),	                // zatial nic, len aby sa dodrzal rom,zone
			(Siz := SIZEOF(NH_ROM_WRK), cfg := 3)	                // 3 = Zone
	        ];
*)
//	aVcf	{HIDDEN}	: ARRAY[1.._Nh_VCF] OF NH_VCF;

END_VAR

(* ---- _Nh_WRK.st ---- *)
{ $IFDEF __NH_WRK }

VAR_GLOBAL                                            // len pre ladenie
   _NhWrk      {HIDDEN} : BOOL := true ;
   { $ IF CPU_CODE > 1999  }
   yIdx         : ARRAY[1..30]	OF NH_IDX;

	yScn			{HIDDEN} : ARRAY[1..50]  OF NH_SCN;
   ypScn 		{HIDDEN} : ARRAY[1..20]  OF NH_SVA_PAR;
	yAct			{HIDDEN} : ARRAY[1..50]  OF NH_ACT;
//	yAla			{HIDDEN} : ARRAY[1..10]  OF NH_ALA;

//		yyVaz	{HIDDEN}	: ARRAY[1.._Nh_VAZ] OF NH_VAZ_CFG ;

		yVaz1			{HIDDEN} : ARRAY[1..50]  OF NH_VAZ;
//	  	yVaz2 		{HIDDEN} : ARRAY[1..150] OF NH_VAZ;
//		yVaz3			{HIDDEN} : ARRAY[1..50]  OF NH_VAZ;
//   	yVaz4			{HIDDEN} : ARRAY[1..80]  OF NH_VAZ;

//  		yGlb			{HIDDEN} : ARRAY[1..1]   OF NH_GLB;
	   yRom			{HIDDEN} : ARRAY[1..30]	OF NH_ROM;
   	yZon			{HIDDEN} : ARRAY[1..10]	OF NH_ROM;
	   ypZon 		{HIDDEN} : ARRAY[1..20]  OF NH_ZON_PAR;
   	yRoW        {HIDDEN} : ARRAY[1..10]  OF NH_WRK_ROM;
		yZoW        {HIDDEN} : ARRAY[1.. 7]  OF NH_WRK_ROM;
		yRol			{HIDDEN} : ARRAY[1..20]  OF NH_ROL;
   	ypRol 		{HIDDEN} : ARRAY[1..100]  OF NH_ROL_PAR;       // 12
//   	yPoi			{HIDDEN} : ARRAY[1..50]  OF NH_POI;

		yTgl			{HIDDEN} : ARRAY[1..30]  OF NH_TGL;
  		ypTgl 		{HIDDEN} : ARRAY[1..120]  OF NH_WSB_PAR;

   ySvd 			{HIDDEN} : ARRAY[1..10]  OF NH_SVD;
   pSvd 			{HIDDEN} : ARRAY[1..100]  OF NH_SVD_PAR;
  	ySva 			{HIDDEN} : ARRAY[1..10]  OF NH_SVA;  //10
  	pSva 			{HIDDEN} : ARRAY[1..40]  OF NH_SVA_PAR;
   yRgb 			{HIDDEN} : ARRAY[1..10]  OF NH_RGB;
	yyRgb 			{HIDDEN} : NH_RGB;
   pRgb 			{HIDDEN} : ARRAY[1..20]  OF NH_RGB_PAR;

	yTve			{HIDDEN} : ARRAY[1..20]  OF NH_TVE;
//	yHet			{HIDDEN} : ARRAY[1..10]  OF NH_HET;  // 20
(*

 	ypHet 		{HIDDEN} : ARRAY[1..20]  OF NH_HET_PAR;       // 10

//	yHev			{HIDDEN} : ARRAY[1..5]   OF NH_HET;  // 20

	yVen 			{HIDDEN} : ARRAY[1..10]  OF NH_TVE;
*)

(*
		yLux			{HIDDEN} : ARRAY[1..5]  OF NH_LUX;
   	yTer 			{HIDDEN} : ARRAY[1..40]  OF NH_TER;
	   yTeh 			{HIDDEN} : ARRAY[1.. 5]  OF NH_TER;
   	yTek 			{HIDDEN} : ARRAY[1.. 5]  OF NH_TER;

*)
//		yRhx			{HIDDEN} : ARRAY[1..2]  OF NH_LUX;
//	yCer			{HIDDEN} : ARRAY[1..3]	 OF NH_TVE;
//	yKot			{HIDDEN} : ARRAY[1..5]	 OF NH_TVE;
//  	yTim			{HIDDEN} : ARRAY[1..10]  OF NH_TIM;
//	yKey			{HIDDEN} : ARRAY[1..3]   OF NH_KEY;

(*
	yDls			{HIDDEN} : ARRAY[1..130]   OF NH_DLS;
	pDls			{HIDDEN} : ARRAY[1..200]   OF NH_RGB_PAR;
	yDlm			{HIDDEN} : ARRAY[1..4]   OF NH_DLM;
	yDlg			{HIDDEN} : ARRAY[1..32]   OF NH_DLG;
*)

//    	yMsg			{HIDDEN} : ARRAY[1..3] OF NH_MSG;

//	  yCat			{HIDDEN} : ARRAY[1..70]	OF NH_CAT;

      yVvo 			{HIDDEN} : ARRAY[1..4]   OF NH_VVO;

   yWsb 			{HIDDEN} : ARRAY[1..30]  OF NH_WSB;
   ypWsb 		{HIDDEN} : ARRAY[1..50]  OF NH_WSB_PAR;

   yTla 			{HIDDEN} : ARRAY[1..10]  OF NH_TLA;

//   ytGl		 {HIDDEN} : ARRAY[1..10]  OF NH_TGL;
//	yPIR			{HIDDEN} : ARRAY[1..50]  OF NH_PIR;
//   ypPir 		{HIDDEN} : ARRAY[1..10]  OF NH_PIR_PAR;

//	yCox			{HIDDEN} : ARRAY[1..10]  OF NH_LUX;

//	yDor			{HIDDEN} : ARRAY[1..10]  OF NH_DOR;

	yFav			{HIDDEN} : ARRAY[1..10]  OF NH_FAV;
   yZas 			{HIDDEN} : ARRAY[1..15]  OF NH_SVD;
   pZas 			{HIDDEN} : ARRAY[1..10]  OF NH_SVD_PAR;
	yyUsr			{HIDDEN} : ARRAY[1..7]   OF NH_USR;

//	ySmw			{HIDDEN} : ARRAY[1..10]  OF NH_SMW;

//	yGat			{HIDDEN} : ARRAY[1.. 5]  OF NH_GAT;
//	yBra			{HIDDEN} : ARRAY[1.. 5]  OF NH_GAT;
//   ypGat 		{HIDDEN} : ARRAY[1..10]  OF NH_GAT_PAR;       // 13

//	ySir			{HIDDEN} : ARRAY[1.. 5]  OF NH_SVD;
//	yBlk			{HIDDEN} : ARRAY[1.. 5]  OF NH_BLK;
//	yBlx			{HIDDEN} : ARRAY[1.. 5]  OF NH_BLX;
//	yBtn			{HIDDEN} : ARRAY[1..20]  OF NH_BTN;
(*
//	yAcl			{HIDDEN} : ARRAY[1..20]  OF NH_VAZ;
*)
//	yVcf			{HIDDEN} : ARRAY[1..150]  OF NH_VAZ_VCF;
//	ySbj			{HIDDEN} : ARRAY[1..4]  OF NH_SBJ;

   { $ ELSE  }

//   	yPoi			{HIDDEN} : ARRAY[1..20]  OF NH_POI;
//	   yRom			{HIDDEN} : ARRAY[1..10]	    OF NH_ROM;
//   	yZon			{HIDDEN} : ARRAY[1..10]	  OF NH_ROM;
//    yRoW        {HIDDEN} : ARRAY[1..10]    OF NH_WRK_ROM;
   { $ END_IF  }

END_VAR

	FUNCTION	_DevDataX {HIDDEN} : BOOL
      VAR_IN_OUT
         aNh   : NH_CFG_CFG;
         dst   : USINT;
      END_VAR
      VAR_INPUT
         n    : UDINT := 10;
      END_VAR
      memsetEx(val := 0,length := n * aNh.Siz , dest := dst ); // vycisti
      IF aNh.Ram > 0 THEN
         MemcpyEx(length := Min(n, INT_TO_UDINT(aNh.Rec)) * aNh.Siz , source := void( mRam[ aNh.Ram ]), dest := dst);
      END_IF;
      _DevDataX := true;
   END_FUNCTION

   FUNCTION	_NhDataWrk {HIDDEN} : BOOL
      VAR_INPUT
         Yes  : BOOL := true ;
      END_VAR
      IF Yes = false THEN
         RETURN;
      END_IF;
		_NhDataWrk :=  TRUE;
      { $ IF CPU_CODE > 1999  }
         { $IFDEF yGlb }
            _DevDataX(aNh := VOID(aCfg[25]), dst := VOID(yGlb), n :=1);
         { $END_IF }
         { $IFDEF yRom }
            _DevDataX(aNh := VOID(aCfg[ 1]), dst := VOID(yrom), n :=30);
         { $END_IF }
         { $IFDEF yPoi }
            _DevDataX(aNh := VOID(aCfg[26]), dst := VOID(yPoi), n := 50);
         { $END_IF }
      { $ ELSE  }
         { $IFDEF yRom }
            _DevDataX(aNh := VOID(aCfg[ 1]), dst := VOID(yrom), n :=10);
         { $END_IF }
         { $IFDEF yPoi }
            _DevDataX(aNh := VOID(aCfg[26]), dst := VOID(yPoi), n := 20);
         { $END_IF }
      { $ END_IF  }

      { $IFDEF yMsg }
      _DevDataX(aNh := VOID(aCfg[46]), dst := VOID(yMsg), n :=3);
      { $END_IF }

      { $IFDEF ycat }
      _DevDataX(aNh := VOID(aCfg[ 2]), dst := VOID(yCat), n :=70);
      { $END_IF }
      { $IFDEF yZon }
      _DevDataX(aNh := VOID(aCfg[ 3]), dst := VOID(yZon), n :=10);
      { $END_IF }
      { $IFDEF ypZon }
      _DevDataX(aNh := VOID(aPar[5]), dst := VOID(ypZon), n :=20);
      { $END_IF }
      { $IFDEF yHet }
      _DevDataX(aNh := VOID(aCfg[ 6]), dst := VOID(yHet));
      { $END_IF }
      { $IFDEF yHev }
      _DevDataX(aNh := VOID(aCfg[47]), dst := VOID(yHev), n:=5);
      { $END_IF }
      { $IFDEF yKot }
      _DevDataX(aNh := VOID(aCfg[ 7]), dst := VOID(yKot), n:=5);
      { $END_IF }
      { $IFDEF ytve }
      _DevDataX(aNh := VOID(aCfg[ 8]), dst := VOID(yTve), n:=20);
      { $END_IF }
      { $IFDEF ycer }
      _DevDataX(aNh := VOID(aCfg[ 9]), dst := VOID(yCer), n := 3);
      { $END_IF }
      { $IFDEF ysvd }
      _DevDataX(aNh := VOID(aCfg[10]), dst := VOID(ySvd));
      { $END_IF }
      { $IFDEF ySva }
      _DevDataX(aNh := VOID(aCfg[11]), dst := VOID(ySva));
      { $END_IF }
      { $IFDEF yVvo }
      _DevDataX(aNh := VOID(aCfg[49]), dst := VOID(yVvo), n :=4);
      { $END_IF }
      { $IFDEF yRgb }
      _DevDataX(aNh := VOID(aCfg[12]), dst := VOID(yRgb));
      { $END_IF }
      { $IFDEF ywsb }
      _DevDataX(aNh := VOID(aCfg[13]), dst := VOID(yWsb), n :=30);
      { $END_IF }
      { $IFDEF ytla }
      _DevDataX(aNh := VOID(aCfg[14]), dst := VOID(yTla));
      { $END_IF }
      { $IFDEF ypir }
      _DevDataX(aNh := VOID(aCfg[15]), dst := VOID(yPir), n :=50);
      { $END_IF }
      { $IFDEF yter }
      _DevDataX(aNh := VOID(aCfg[16]), dst := VOID(yTer), n :=40);
      { $END_IF }
      { $IFDEF yteh }
      _DevDataX(aNh := VOID(aCfg[17]), dst := VOID(yTeh), n := 5);
      { $END_IF }
      { $IFDEF ytek }
      _DevDataX(aNh := VOID(aCfg[18]), dst := VOID(yTek), n := 5);
      { $END_IF }
      { $IFDEF ylux }
      _DevDataX(aNh := VOID(aCfg[19]), dst := VOID(yLux), n := 5);
      { $END_IF }
      { $IFDEF yRhx }
      _DevDataX(aNh := VOID(aCfg[51]), dst := VOID(yRhx), n := 2);
      { $END_IF }
      { $IFDEF yfav }
      _DevDataX(aNh := VOID(aCfg[20]), dst := VOID(yFav));
      { $END_IF }
      { $IFDEF yzas }
      _DevDataX(aNh := VOID(aCfg[21]), dst := VOID(yZas), n:=15);
      { $END_IF }
      { $IFDEF yDor }
      _DevDataX(aNh := VOID(aCfg[33]), dst := VOID(yDor));
      { $END_IF }
      { $IFDEF yyUsr }
      _DevDataX(aNh := VOID(aCfg[22]), dst := VOID(yyUsr), n:=7);
      { $END_IF }
      { $IFDEF yven }
      _DevDataX(aNh := VOID(aCfg[23]), dst := VOID(yVen));
      { $END_IF }
      { $IFDEF yKey }
      _DevDataX(aNh := VOID(aCfg[24]), dst := VOID(yKey), n := 3);
      { $END_IF }
      { $IFDEF ysmw }
      _DevDataX(aNh := VOID(aCfg[45]), dst := VOID(ySmw));
      { $END_IF }
      { $IFDEF yRol }
      _DevDataX(aNh := VOID(aCfg[31]), dst := VOID(yRol), n:=20);                    //ROL
      { $END_IF }
      { $IFDEF yBra }
      _DevDataX(aNh := VOID(aCfg[37]), dst := VOID(yBra), n := 5);            //BRA - stara
      { $END_IF }
      { $IFDEF yGat }
      _DevDataX(aNh := VOID(aCfg[37]), dst := VOID(yGat), n := 5);            //BRA
      { $END_IF }
      { $IFDEF ySir }
      _DevDataX(aNh := VOID(aCfg[32]), dst := VOID(ySir), n := 5);            //SIR
      { $END_IF }
      { $IFDEF yBlk }
      _DevDataX(aNh := VOID(aCfg[35]), dst := VOID(yBlk), n := 5);            //BLK
      { $END_IF }
      { $IFDEF yBlx }
      _DevDataX(aNh := VOID(aCfg[36]), dst := VOID(yBlX), n := 5);            //BLK
      { $END_IF }
      { $IFDEF yTgl }
      _DevDataX(aNh := VOID(aCfg[40]), dst := VOID(yTgl), n :=30);
      { $END_IF }
      { $IFDEF yBtn }
      _DevDataX(aNh := VOID(aCfg[41]), dst := VOID(yBtn), n := 20);
      { $END_IF }
      { $IFDEF yDlm }
      _DevDataX(aNh := VOID(aCfg[42]), dst := VOID(yDlm), n := 4);
      { $END_IF }
      { $IFDEF yDls }
      _DevDataX(aNh := VOID(aCfg[43]), dst := VOID(yDls), n := 130);
      { $END_IF }
      { $IFDEF yDlg }
      _DevDataX(aNh := VOID(aCfg[44]), dst := VOID(yDlg), n := 32);
      { $END_IF }
      { $IFDEF yTim }
      _DevDataX(aNh := VOID(aCfg[50]), dst := VOID(yTim), n := 10);
      { $END_IF }
      { $IFDEF yScn }
      _DevDataX(aNh := VOID(aCfg[ 4]), dst := VOID(yScn), n := 50);
      { $END_IF }
      { $IFDEF yact }
      _DevDataX(aNh := VOID(aCfg[ 5]), dst := VOID(yAct), n:= 50);
      { $END_IF }
      { $IFDEF yAla }
      _DevDataX(aNh := VOID(aCfg[48]), dst := VOID(yAla));
      { $END_IF }
      { $IFDEF yVaz1 }
      _DevDataX(aNh := VOID(aVaz[ 1]), dst := VOID(yVaz1), n := 50);
      { $END_IF }
      { $IFDEF yVaz2 }
      _DevDataX(aNh := VOID(aVaz[ 2]), dst := VOID(yVaz2), n :=150);
      { $END_IF }
      { $IFDEF yVaz3 }
      _DevDataX(aNh := VOID(aVaz[ 3]), dst := VOID(yVaz3), n := 50);
      { $END_IF }
      { $IFDEF yVaz4 }
      _DevDataX(aNh := VOID(aVaz[ 4]), dst := VOID(yVaz4), n :=80);
      { $END_IF }

(*
      { $IFDEF yAcl }
      _DevDataX(aNh := VOID(aVaz[ 5]), dst := VOID(yAcl), n := 20);
      { $END_IF }
*)

      { $IFDEF pSvd }
       _DevDataX(aNh := VOID(aPar[1]), dst := VOID(pSvd), n := 100);
      { $END_IF }
      { $IFDEF pSva }
      _DevDataX(aNh := VOID(aPar[2]), dst := VOID(pSva), n := 40);
      { $END_IF }
      { $IFDEF pRgb }
      _DevDataX(aNh := VOID(aPar[3]), dst := VOID(pRgb), n:=20);
      { $END_IF }
      { $IFDEF ypWsb }
      _DevDataX(aNh := VOID(aPar[4]), dst := VOID(ypWsb), n := 50);
      { $END_IF }
      { $IFDEF ypTgl }
      _DevDataX(aNh := VOID(aPar[15]), dst := VOID(ypTgl), n := 120);
      { $END_IF }
      { $IFDEF pTla }
      _DevDataX(aNh := VOID(aPar[5]), dst := VOID(ypTla), n:=20);
      { $END_IF }
      { $IFDEF pZas }
      _DevDataX(aNh := VOID(aPar[6]), dst := VOID(pZas));
      { $END_IF }
      { $IFDEF ypPir }
      _DevDataX(aNh := VOID(aPar[7]), dst := VOID(ypPir));
      { $END_IF }
      { $IFDEF ypHEt }
      _DevDataX(aNh := VOID(aPar[9]), dst := VOID(ypHet), n := 20);
      { $END_IF }
      { $IFDEF ypScn }
      _DevDataX(aNh := VOID(aPar[10]), dst := VOID(ypScn), n := 20);
      { $END_IF }
      { $IFDEF ypRol }
      _DevDataX(aNh := VOID(aPar[12]), dst := VOID(ypRol), n:=100);
      { $END_IF }
      { $IFDEF ypGat }
      _DevDataX(aNh := VOID(aPar[13]), dst := VOID(ypGat));
      { $END_IF }
      { $IFDEF yCox }
      _DevDataX(aNh := VOID(aCfg[41]), dst := VOID(yCox), n :=10);
      { $END_IF }
      { $IFDEF pDls }
      _DevDataX(aNh := VOID(aPar[16]), dst := VOID(pDLs), n := 200);
      { $END_IF }

// WRK
      { $IFDEF yCaW }
//         memset(val := 0, length := aSys.sCaW, dest := VOID( mRam[aSys.aCaW1] ));
         MemcpyEx(length :=  aSys.sCaW  , source := void( mRam[aSys.aCaW1] ), dest := VOID(yCaW));
      { $END_IF }
      { $IFDEF yRoW }
         MemcpyEx(length :=  MIN(10,aSys.sRoW/SIZEOF(NH_WRK_ROM))  , source := void( mRam[aSys.aRoW1] ), dest := VOID(yRoW));
      { $END_IF }
      { $IFDEF yZoW }
         MemcpyEx(length :=  MIN( 7,aSys.sRoW/SIZEOF(NH_WRK_ROM))  , source := void( mRam[aSys.aZoW1] ), dest := VOID(yZoW));
      { $END_IF }

      { $IFDEF yIdx }
         memset(val := 0, length := 30 * SIZEOF(NH_IDX), dest := VOID(yIdx));
         MemcpyEx(length :=  MIN(30,USINT_TO_UDINT(aWeb.M[1].ixb[0].idx + aWeb.M[1].ixb[1].idx)) * SIZEOF(NH_IDX)  , source := void( mRam[aSys.vIx1] ), dest := VOID(yIdx));
      { $END_IF }

   END_FUNCTION

{ $ ELSE }
   VAR_GLOBAL                                            // len pre ladenie
      _NhWrk      {HIDDEN} : BOOL := false;
   END_VAR
{ $END_IF }

(* ---- _Nh_Frm_BRW.st ---- *)
FUNCTION _Nh_Frm_Row_BRW {HIDDEN}    : BOOL        // naplni, alebo refreshne objekty jedneho riadka browsu/frame/home
	{ $ IFDEF __NH_WEB }
   VAR_INPUT
      new   : BOOL;
      row   : USINT;
   END_VAR
   VAR_TEMP
		blk	: USINT;
      cp    : USINT;
//      np    : INT;
   END_VAR
   _Nh_Frm_Row_BRW := true;
   IF new THEN
		cp := xR^.h.cf.c;
      IF xL^.obj = 11 AND xR^.h.cf.c = 1 THEN                                           // ZONA domcek       1 ZON -> ROMs
			cp := 3;
		ELSIF xR^.h.new  THEN
			new := false;
      END_IF;
		IF new THEN
      	_Nh_Brw_Row_DSH(row := row, frm := USINT_TO_UINT(aCfg[ cp ].fBr) );   	// nacita FRM a podla DSH pripravi korekcie X,Y
			_Nh_Brw_Row_OBJ(row := row);
	      _Nh_FRM_Read(frm:=246);   	// nacita rozne preddefinovane objekty v riadku	 xR^.o.ob[]
	     	_Nh_Chk_FAV();
   	   CASE xR^.h.cf.c OF
			 0:	;
			50:	// timer - v priebehu refreshu sa nemeni
					xTim	:= xDev;
					memcpyPTR(length:=SIZEOF(NH_OBJ_DAT), source:=ADR(yFrm_246.tim_1), dest:=ADR(xR^.o.ob[6]) );		// nastavi zobrazovanie obrazka typu casovaca nad hlavnou ikonou
					memcpyPTR(length:=SIZEOF(NH_OBJ_DAT), source:=ADR(yFrm_246.e4O1), dest:=ADR(xR^.o.ob[7]) );		// vypne zobrazovanie na stavovou ikonou
			 		x4o   			:= ADR(xR^.o.ob[6]);
					x4o^.obr[2]    :=	yFrm_246.tim_1_typ_obr[ xTim^.cf.typ ];			// podla typu vyberie obrazok
					blk	:= 5;
	      END_CASE;

	   END_IF;
	END_IF;

   CASE xR^.h.cf.c OF

   	0: ;
    	1:	_Nh_Shw_ROM_ROW();
		2: // CAT
		   	_Nh_FRM_Read(frm:=232);
            xR^.o.ob[5].cf.c := 0;
  	         xR^.o.ob[5].cf.n := yFrm_232.cat[xR^.h.cf.n].txt;                                  // cislo textu v 1.riadku
            xR^.o.ob[6].cf.c := 0;
  	         xR^.o.ob[6].cf.n := yFrm_232.cat[xR^.h.cf.n].txt+1;                                  // cislo textu v 2.riadku je za prvym
				IF yFrm_232.cat[xR^.h.cf.n].cmd4 = 0 THEN
					xR^.o.ob[4].wh := 0;
				ELSE
					xR^.o.ob[4].cm := yFrm_232.cat[xR^.h.cf.n].cmd4;
				END_IF
				IF yFrm_232.cat[xR^.h.cf.n].cmd2 = 0 THEN
					xR^.o.ob[2].wh := 0;
				ELSE
					xR^.o.ob[2].cm := yFrm_232.cat[xR^.h.cf.n].cmd2;
				END_IF
				xR^.o.ob[1].cm := yFrm_232.cat[xR^.h.cf.n].cmd1;

            IF xA^.usr= 1 THEN                                                   // pre admina vypise cislo CAT
               xR^.o.ob[7].wh    := 6;
               xR^.o.ob[7].cf.c  := 254;
               xR^.o.ob[7].fmt   := CONCAT(INT_TO_STRINGF(xR^.h.cf.n,'%2u'), '');
            END_IF;
		3:	xR^.o.ob[9].cf.c:=252;										// vypisuje sa nazov domceka (domovskej zony)
				_Nh_Shw_ROM_ROW();
		6: // HET
  				xHet  	:= xDev;
				IF xL^.dsh = 4 THEN
					_Nh_Shw_CPY();
      		ELSE
					_NH_Het_Map_Reg();
//					IF xHet^.io[0].own THEN                // DEV regulovanej teploty
               	IF xRegMod^.wht = 1 THEN
							xR^.o.ob[2].fmt := REAL_TO_STRINGF(xHet^.al.ou.val,'%5.1f°');
						ELSE
							xR^.o.ob[2].fmt := REAL_TO_STRINGF(xHet^.al.ou.val,'%5.0f %%');
						END_IF
//					END_IF ;
					IF xHet^.io[1].own THEN                // ma termoventil
						IF xHet^.io[1].zon THEN             // TVE ma teplotu
							xR^.o.ob[5].fmt := REAL_TO_STRINGF(xHet^.io[1].val,'%5.1f°');
						ELSE
						   xR^.o.ob[5].wh := 0;
						END_IF;
						xHet^.al.lst := true;
					ELSE
		   			xR^.o.ob[5].wh := 0;
						xHet^.al.lst := false;
					END_IF;
//	 			IF xA^.admin = false THEN
	 				IF xM^.set=false OR xA^.UsrRight < 2 THEN
	 					xR^.o.ob[1].cm   := 0;
 						xR^.o.ob[4].fn   := 0;
 						xR^.o.ob[6].fn   := 0;
					END_IF;
				END_IF;
  		47: // HEV
            xHet  := xDev;
				IF xL^.dsh = 4 THEN
					_Nh_Shw_CPY();
         	END_IF;
      		IF xHet^.io[0].own THEN                // aktualne % CO2 zo snimaca
					xR^.o.ob[2].fmt := REAL_TO_STRINGF(xHet^.io[0].val,'%6.0f %%');
				END_IF;
				IF xHet^.io[2].own THEN                // ma termoventil
					xHet^.al.lst := true;
				ELSE
					xHet^.al.lst := false;
				END_IF;
//  	 			IF xA^.admin = false THEN
	 			IF xM^.set=false OR xA^.UsrRight < 2 THEN
 					xR^.o.ob[1].cm   := 0;
	 				xR^.o.ob[4].fn   := 0;											// setup nie je
 					xR^.o.ob[6].fn   := 0;                               	// lst vazby nie su
  				END_IF;
				IF xL^.chk AND xR^.o.ob[4].cf.c > 0 THEN
					IF acfg[xR^.o.ob[4].cf.c].tgrp = 15 THEN
 						xR^.o.ob[7].wh   := 0;                      			// ked je vo vazbe PIR, vypnu sa predvolby a zobrazuju sa prvky PIR
					END_IF;
				END_IF;

		7: // KOT
 			_Nh_Shw_TVE_ROW();

		8: // TVE
 			_Nh_Shw_TVE_ROW();

		9: // CER
 			_Nh_Shw_TVE_ROW();

		15: //PIR
				IF	xR^.h.pir THEN					// je vo vazbe
					;
				ELSIF	_NhxRom(nr := xDev^.cf.rom ,x:=55) THEN
					_Nh_Shw_107_ROM(o:=7, day:=true);
	            _Nh_Frm_STA_OU(obj:=2, o:=8);
					blk	:= 5;
//   				_Nh_DEF_VAR(wh:=20, o:=6, x:=ADR(xDev^.cf.blk) );
				ELSE
					xR^.o.ob[7].wh		:= 0;
				END_IF;

		23: // REK
				 _Nh_Shw_TVE_ROW();

		31: // ROL
				xRol 		:= xDev;
				IF new  THEN                        // pri prvom vstupe do FRM. nacitat iny formular podla menu. n
					xRo		:= ADR(xR^.o.ob[5]);
					IF xR^.h.cf.p=0 THEN
						xR^.h.cf.p := xRol^.cf.par;
					END_IF;
					xRo^.cf	:= xR^.h.cf;
					xRo^.chk	:= xL^.chk;					// priznak vazby
				END_IF;

  	 			IF xM^.set AND xF^.cf.c = 2 AND xF^.cf.n = 3 THEN		// pristupne kopirovanie
		  	 			IF xU^.o[1].fn  = 44 AND xL^.dsh = 1 THEN									// zlte COPY
//      D1_7       : NH_OBJ_4O1 	:= (obj:=1, obr:=[44,38,0,0], cmd:=[0,0,0,0], wxy:=[0,0,0,0],ok:=[0,0,0,0], txt:=[0,0,0,0],  );                          // 5=slider;
//							xR^.o.ob[7]		:= xR^.o.ob[8];
						 	x4o    			:= ADR(xR^.o.ob[8]);
							xR^.o.ob[1].cm 	:= 128;									// click na hlavnu ikonu = oznacovanie
							xR^.o.ob[10].cm 	:= 128;									// nazov
							x4o^.wh			:= 107;
							x4o^.obj			:= 1;
   	 					x4o^.wxy[1]    := 52;
    						x4o^.wxy[2]    := 42;
							x4o^.obr[1]		:= 44;
							x4o^.obr[2]		:= 38;
							x4o^.ok[1] 		:= xU^.o[1].wh = xR^.h.cf.n;
							x4o^.ok[2] 		:= xRol^.me.cpy;
						ELSE
							xR^.o.ob[1].cm 	:= 204;                         	// standardne parametre rolety
							xR^.o.ob[10].cm 	:= 204;								// nazov
							x4o^.wh				:= 0;
						END_IF;
				END_IF;

		131: // ROL
            xRol     := xDev;
				IF new THEN
	            ix       := xR^.o.ob[6].fn;                                             // slider je v 8
   	         xS       := ADR(xB^.s[ix]);
		         _NhSetObjBrw(ob:=5, wh:=24, w:=50,  t:=4, c:=1, cm:=48,  vb := ADR(xRol^.cx.SetLam),   fmt := '119500');        // ROL/LAM
         	   _Nh_Frm_Row_O13(ob:=6, vb:= PTR_TO_UDINT( ADR(xRol^.al.in.Val) ) );
	  	 			IF xM^.set AND xF^.cf.c = 2 AND xF^.cf.n = 3 THEN		// pristupne kopirovanie
		  	 			IF xU^.o[1].fn  = 44 THEN									// zlte COPY
//      D1_7       : NH_OBJ_4O1 	:= (obj:=1, obr:=[44,38,0,0], cmd:=[0,0,0,0], wxy:=[0,0,0,0],ok:=[0,0,0,0], txt:=[0,0,0,0],  );                          // 5=slider;
							xR^.o.ob[7]		:= xR^.o.ob[8];
						 	x4o    			:= ADR(xR^.o.ob[7]);
							xR^.o.ob[1].cm := 128;									// click na hlavnu ikonu = oznacovanie
							x4o^.wh			:= 107;
							x4o^.obj			:= 1;
   	 					x4o^.wxy[1]    := 52;
    						x4o^.wxy[2]    := 42;
							x4o^.obr[1]		:= 44;
							x4o^.obr[2]		:= 38;
							x4o^.ok[1] 		:= xU^.o[1].wh = xR^.h.cf.n;
							x4o^.ok[2] 		:= xRol^.me.cpy;
						ELSE
							xR^.o.ob[1].cm := 204;                         	// standardne parametre rolety
							x4o^.wh			:= 0;
						END_IF;
					END_IF;
				 	x4o    			:= ADR(xR^.o.ob[8]);
					x4o^.wh			:= 107;
					y4o := x4o^;
					IF xRol^.cx.yLam <= 0.0 THEN
						x4o^.obr[1]		:= 500;
					ELSIF xRol^.cx.yLam >= 100.0 THEN
						x4o^.obr[1]		:= 502;
					ELSE
						x4o^.obr[1]		:= 501;
					END_IF;
					IF xRol^.cx.CMD = 12 THEN
						x4o^.ok[2]		:= true;										// zobrazi blokovanie vetrom
					ELSE
						x4o^.ok[2]		:= false;
					END_IF;

//					x4o^.obr[1]		:= 10000+REAL_TO_INT(xRol^.cx.yBli);			// namiesto obr sa vypise text = poziacia rolety
//					x4o^.obr[3]		:= 10000+REAL_TO_INT(xRol^.cx.yLam);			//

				END_IF;
				IF xRol^.cx.SetLam = false THEN								// slider ROL
//    				xR^.o.ob[6].BgC := 9;                              // modra
    				xR^.o.ob[6].BgC := 3;                              // modra
					IF xRol^.cx.CMD > 200 THEN
						xRol^.al.in.Val := xRol^.cx.yrol;
					END_IF;
				ELSE
//					xR^.o.ob[6].BgC := 10;                                	// biela pre LAM
					xR^.o.ob[6].BgC := 27;                                	// biela pre LAM
					IF xRol^.cx.CMD > 200 THEN
						xRol^.al.in.Val := xRol^.cx.yLam;
					END_IF;
         	END_IF;

		37: // GATE
				xGat	:= xDev;
            xR^.o.ob[5].fn := _Nh_O12(xGat^.cx.btn,69,66);                   // slider - aktivovana SCN je oranzova, inak zlta
				IF  xGat^.cf.typ < 2 THEN											// garaz,brana
					_Nh_Frm_Row_O13(ob:=6, t:=0, vb:=PTR_TO_UDINT( ADR(xDev^.al.ou.val) ));
				ELSE
					xR^.o.ob[6].wh := 0;
				END_IF;
				_Nh_Frm_STA_OU(obj:=2, o:=8);

		{$IFDEF __NH_DALI}
		42: // DL-M
   	         xDlm              := xDev;
      	      ix                := xR^.h.cf.n;
         	   xDLfb             := ADR(aDali[ix]) ;
	            _Nh_Frm_Row_O13(ob:=5);

//    				xB^.s[ 0 ].v2 := 254.0;                         // ine ako DALI maju max 100%

   	         xPtD              := ADR(xR^.o.ob[9].cf.n);
      	      xPtD^             := PTR_TO_UDINT( ADR(xDlfb^.txt) );                   // v druhom riadku sa zobrazuje INFO o aktualnom parametre
         	   xR^.o.ob[9].cf.c  := 253;                                               // hodnota v pointri
(*
            xR^.o.ob[8].fmt   := INT_TO_STRING(xR^.h.cf.n);                         // cislo DLM l hlavnej ikone
            xR^.o.ob[8].BgC   := _Nh_U12(xDlm^.cx.sta.Present,8,1);                 // vykonany random/nevykonany
            xR^.o.ob[7].wh    := 0;
*)
	            xR^.o.ob[4].fn := _Nh_O12(xDlm^.cx.dlm.nShA>0,25,23 );                  // zeleny/sivy setup
//            xR^.o.ob[6].fn := _Nh_O12(xDLm^.al.lst,334,333);                  		// zeleny/sivy setup

      	      IF xDLm^.cx.sta.Err  THEN
         	      xDlfb^.txt := CONCAT(xDlfb^.txt,' E:');
            	   xDlfb^.txt := CONCAT(xDlfb^.txt,' '
               	                                                                     // RndAdr               Query
                  	                  ,USINT_TO_STRING(xDLm^.me.err.nErrS[1]),';'     // neprisla odpoved     Neprisla odpoved
                     	               ,USINT_TO_STRING(xDLm^.me.err.nErrS[2]),';'     // kolizia adries       Kolizia 2 adries
                        	            ,USINT_TO_STRING(xDLm^.me.err.nErrS[3]),';'     // niet co hladat
                           	         ,USINT_TO_STRING(xDLm^.me.err.nErrS[4]) );
	               xDlfb^.txt := CONCAT(xDlfb^.txt,'/'
   	                                 ,USINT_TO_STRING(xDLm^.me.err.nErrG[1]),';'
      	                              ,USINT_TO_STRING(xDLm^.me.err.nErrG[2]),';'
         	                           ,USINT_TO_STRING(xDLm^.me.err.nErrG[3]),';'
            	                        ,USINT_TO_STRING(xDLm^.me.err.nErrG[4]) );

//					ELSIF xDLfb^.cmd[1].cmd = 0 THEN
//	   	         xDlfb^.txt        := USINT_TO_STRINGF(xDlm^.cx.dlm.nSha,'%2d');         // pocet SHA
					ELSE
//	   	         xDlfb^.txt        := USINT_TO_STRINGF(xDlfb^.cmdQue,'%2u');         // pocet SHA
	            END_IF;
   	         // skupina
      	      // nazov DLM
         	   xR^.o.ob[10].cf   := xR^.h.cf;
	            x4o            := ADR(xR^.o.ob[7]);
   	         x4o^.obr[1]   := USINT_TO_INT( xDlm^.cx.dlm.nShA );
      	      IF xDLm^.cx.sta.Present = false THEN
         	      x4o^.BgC[1] := 2;
	            ELSE
   	            x4o^.BgC[1] := 3;
      	      END_IF;
		         x4o^.ok[2]        := 1;
      	      x4o^.obr[2]       := xR^.h.cf.n;

	            IF xDLm^.me.err.nErrS[2] > 0 THEN
   	            x4o^.ok [3] := 1;
      	         x4o^.obr[3] := USINT_TO_INT( xDLm^.me.err.nErrS[2] );
         	   ELSE
            	   x4o^.ok[3]        := 0;
	            END_IF;

      43: 	// DLS
    	      // xL^.obj :
				// 47 DLm/DLg
				// 48 DLm/DLs

				// 43 v hlavicke je toto 	DLs riadok je DLg 		priradzuje sa DLs->DLg
				// 44 v hlavicke je 			DLg riadok je toto DLs  priradzuje sa DLs->DLg
				xDLs     := xDev;
	         dlsl     := _Nh_DL_sha(nd := xR^.h.cf.n);
   	      dlma     := _Nh_DL_sha(ma := true, nd := xR^.h.cf.n);
				IF new THEN
	            x4o   := ADR(xR^.o.ob[7]);
					IF xM^.set AND xA^.UsrRight > 2 THEN
						x4o^.wh			:= 107;
	   	         x4o^.obr[1]   	:= USINT_TO_INT( dlsl );
  	      	      IF xDLs^.cx.sta.Present = false THEN
     	      	      x4o^.BgC[1] := 2;
      	         ELSE
  	      	         x4o^.BgC[1] := 5;
     	      	   END_IF;
        	      	IF xDLs^.cx.sta.ErrID > 0 THEN
           	      	x4o^.ok [3] := 1;
               	   x4o^.obr[3] := USINT_TO_INT( xDLs^.cx.sta.ErrID );;
	                  xR^.o.ob[0].FgC := 7;                                 				// cela dlazdica bude cevena
  		            ELSE
     		            x4o^.ok[3]        := 0;
        		         xR^.o.ob[0].FgC   := 1;
           		   END_IF;
	               x4o^.ok[2]  := 1;
  		            x4o^.obr[2] := USINT_TO_INT( dlma );

						IF xR^.h.chk  = false  THEN                                 		// len ked nie je vo vazbach
							xR^.o.ob[5].w  	:= 300;        											// skrati slider {mozno ho out5inOne aj tak prepise}
							xR^.o.ob[6] 		:= _NhBrwObj.dlgl;										// obrazok vseobecneho listu
							IF xDLs^.cx.scn.grp<>_eBtn15 THEN
  	   						xR^.o.ob[6].fn   	:= 334;
							ELSIF xDev^.al.lst THEN
     							xR^.o.ob[6].fn   	:= 192;
							ELSE
     							xR^.o.ob[6].fn   	:= 39;
							END_IF;
						END_IF;
					ELSE
						x4o^.wh			:= 0;
					END_IF;

						IF xDls^.cx.cfg.out5inOne THEN
							xR^.o.ob[5] 		:= _NhBrwObj.rgbwa;										// RGBWA namiesto slidera
							xR^.o.ob[5].wh		:= 121;
							xR^.o.ob[4].fn		:= 124;
							xR^.o.ob[4].cm		:= 74;	                                       // otvori priradenie RGBWA k DEV
							xR^.o.ob[2].cm 	:= 249;														// posle prikaz ON/OFF pre 5in1, hoci je aj chk
						END_IF;

					IF xR^.h.chk THEN
						_NhxPt(c := xF^.cf.c, n := xF^.cf.n,x:=432);
						IF xF^.cf.c = 44 THEN                                			// do DLg
							// DLs v scene nema parameter, nastavuje sa len LVL v strukture
	     					dlgr := _Nh_DL_sha(gr:=1,nd := xF^.cf.n)-100 ;				// 0..15
							_Nh_Frm_Row_O13(ob:=5, t:=1, vb:=PTR_TO_UDINT(ADR(xDLs^.cx.scn.LVL[ dlgr ])) );
							xR^.o.ob[2].cm 	:= 0;
						ELSIF xDls^.cx.cfg.out5inOne THEN
							IF xF^.cf.c = 8 THEN													// zatial len pre TVE
								xR^.o.ob[6] 		:= _NhBrwObj.srgbwa;							// led na sebe = ktory port {RGBWA} je priradeny k DEV v hlavicke
								xR^.o.ob[6].cm 	:= 251;											// posle prikaz ON/OFF pre 5in1
								_NhxPt(c:=xF^.cf.c, n:=xF^.cf.n, x:=-154);
								xTve := xPt;
								_Nh_DEF_VAR(wh:=20, o:=6, x:=ADR(xTve^.io[0].dev.o));
							ELSE
								xR^.o.ob[6].wh 	:= 0;											// nebude zobrazovat vyber konkretnej farby
							END_IF;
						ELSIF _Nh_IO_MAP(cIo:=xF^.cf.c, Dev:=xR^.h.cf.c)  THEN
							_Nh_Frm_Row_O13(ob:=5, t:=0, vb:=PTR_TO_UDINT(ADR( xPtIOa^.val ) ));
							xR^.o.ob[2].cm 	:= 0;
						ELSIF xR^.o.ob[4].cf.c = 15 THEN                                				// check PIR ma prednost
      					xR^.o.ob[5].wh 	:= 0;
						ELSIF _NhxPar(cp := aCfg[xR^.h.cf.c].par , np := xR^.h.cf.p,x:=-1006) THEN		// SCN,ACT,BLK
							_Nh_Frm_Row_O13(ob:=5, t:=1, vb:=PTR_TO_UDINT(ADR(xPar^.all.lvl)) );
						ELSE
							xR^.o.ob[5].wh := 0;
							xR^.o.ob[2].cm := 0;
						END_IF;

(*
					ELSIF xDls^.cx.cfg.out5inOne THEN								// do TVE, bude zobrazena RGBWA +
						xR^.o.ob[5] 		:= _NhBrwObj.rgbwa;											// obrazok vseobecneho listu
						xR^.o.ob[5].wh		:= 121;
						xR^.o.ob[2].cm 	:= 249;													// posle prikaz ON/OFF pre 5in1
*)
					END_IF;

				ELSIF	xR^.h.chk THEN
						IF xF^.cf.c = 44 THEN                                		// do DLg
      					dlgr := _Nh_DL_sha(gr:=1,nd := xF^.cf.n)-100 ;				// 0..15
							IF  xR^.o.ob[2].tch THEN												// prepnut LVL s status - LVL je uz zapisany v parametri
								xDLs^.cx.scn.LVL[ dlgr ] := xPar^.all.lvl;
							END_IF;
							IF xR^.o.ob[2].tch OR (xR^.o.ob[5].tch AND xA^.tch.Qf) THEN
//		                  _Nh_DL_ADD_Task(wht:=  4, par:= 1, sha := dlsl , val := dlGr+100, dlm := dlma  );	// prida ballast do sceny, hoci tam uz moze byt
//      		            _Nh_DL_ADD_Task(wht:=102, par := dlgr,  	//   scena		0..15                    	// nastavi LVL pre ballast v scene
      		            _Nh_DL_ADD_Task(wht:=2, par := dlgr,  	//   scena		0..15                    	// nastavi LVL pre ballast v scene
         	                                   	sha := dlsl,    //   ballast	0..63
            	                                	val := REAL_TO_USINT(USINT_TO_REAL(xDLs^.cx.scn.LVL[ dlgr ])*2.45) ,
               	                             	dlm := dlma );
							END_IF;
						END_IF;
				ELSIF xDls^.cx.cfg.out5inOne THEN								// do TVE, bude zobrazena RGBWA +
					;
//					xR^.o.ob[4].fn	:= 124;
//					xR^.o.ob[4].cm	:= 76;

				ELSE
					_Nh_Frm_Row_O13(ob:=5, t:=0, vb:=PTR_TO_UDINT(ADR(xDev^.al.in.val)) );
				END_IF;

				IF xDls^.cx.cfg.out5inOne THEN
						;
				ELSE
					_Nh_Frm_STA_OU(obj:=2, o:=8);											// ikony nad stavovym obrazkom
				END_IF;

      44: // DLg
			      // 56:  DLs ->  DLg		... v hlavicke je DLsa v riadkoc su sceny do ktorych moze ist
				   xDLg     := xDev;
   	         dlma     := _Nh_DL_sha(gr:=1, ma := true, nd := xR^.h.cf.n);            // master
      	      dlgr     := _Nh_DL_sha(gr:=1, nd := xR^.h.cf.n)-100;                    // cislo GRP - 100 prevedie na 0..15
					xDLg^.al.lst	:= xDLg^.cx.Sta.Present;											// dolezitejsi je Present, je aj po restarte aktivny
	            x4o   := ADR(xR^.o.ob[7]);
       			IF xR^.h.chk  THEN
						IF xF^.cf.c = 43  THEN																// DLs v hlavicke do tejto sceny
							IF _NhXPt(c:=xF^.cf.c, n:=xF^.cf.n,x:=-135) THEN
								xDLs := xPt;
					         dlsl     := _Nh_DL_sha(nd := xF^.cf.n);
								_Nh_Frm_Row_O13(ob:=5, t:=1, vb:=PTR_TO_UDINT(ADR(xDLs^.cx.scn.lvl[dlgr])) );
								IF (xR^.o.ob[5].tch AND xA^.tch.Qf) THEN
      			            _Nh_DL_ADD_Task(wht:=2,par := dlgr,  	//   scena		0..15                    	// nastavi LVL pre ballast v scene
         		                                   sha := dlsl,    //   ballast	0..63
            		                                val := REAL_TO_USINT(USINT_TO_REAL( xDLs^.cx.scn.LVL[ dlgr ])*2.45),
               		                             dlm := dlma );
								END_IF;
							ELSE
								xR^.o.ob[5].wh := 0;
							END_IF;
						ELSIF xR^.o.ob[4].cf.c <>  15 THEN
		         	   _Nh_Frm_Row_O13(off:=xR^.h.pir, ob:=5);
						END_IF;

					ELSE
	         	   _Nh_Frm_Row_O13(off:=xR^.h.pir, ob:=5);
//		            xR^.o.ob[5].BgC := _Nh_U12(xDLg^.al.ou.val=254.0,6,5);                   // slider - aktivovana SCN je oranzova, inak zlta
		            xR^.o.ob[5].BgC := _Nh_U12(xDLg^.al.ou.val=100.0,6,5);                   // slider - aktivovana SCN je oranzova, inak zlta
					END_IF;

					IF xM^.set AND xA^.UsrRight > 2 THEN
							x4o^.wh	:= 107;
      		         x4o^.obr[1]   := USINT_TO_INT( dlgr );
         		      IF xDLg^.cx.sta.Present = false THEN
            		      x4o^.BgC[1] := 2;
	          	     	ELSE
   	         	      x4o^.BgC[1] := 6;
	   	            END_IF;
   	   	         IF xDLg^.cx.sta.ErrID > 0 THEN
      	   	         x4o^.ok [3] := 1;
         	   	      x4o^.obr[3] := USINT_TO_INT( xDLg^.cx.sta.ErrID );;
            	   	   xR^.o.ob[0].FgC := 7;                                 // cela dlazdica bude cevena
	               	ELSE
		                  x4o^.ok[3]        := 0;
   		               xR^.o.ob[0].FgC   := 1;
      		         END_IF;
         		      x4o^.ok[2]  := 1;
            		   x4o^.obr[2] := USINT_TO_INT( dlma );

                  IF xR^.o.ob[4].cf.c = 15 THEN
   			         xR^.o.ob[5].wh 	:= 0;
						ELSIF xR^.o.ob[6].wh <> 1 THEN
   						xR^.o.ob[6] 		:= _NhBrwObj.list;											// obrazok vseobecneho listu
	     	            xR^.o.ob[6].fn   	:= _Nh_O12(in := xDev^.al.lst , o1:=192, o2:=39); // LIST zeleny/sivy
						   xR^.o.ob[5].w  	:= 300;        												// skrati slider
						END_IF;

   				ELSE
						x4o^.wh	:= 0;
   				END_IF;

(*
					IF NOT( xR^.o.ob[4].cf.c = 15 AND xR^.h.chk ) THEN
						xR^.o.ob[6].wh	:= 1;															// ked je vo vazbe PIR
   				END_IF;
*)
      	      IF xDlg^.cf.rom = 0 THEN
         	      xR^.o.ob[9].wh := 0;
	            END_IF;
            	// 53 DLs/DLg
					_Nh_Frm_STA_OU(obj:=2, o:=8);

		{$ELSE}
	        	42: // DL-M
					;
  				43: // DLS
					;
	        	44: // DL-M
					;
		{$END_IF}

	  48:	// ALA
   		xAla  := xDev;
   		_NhxZon(nz:=xAla^.cf.rom);
	   	xR^.o.ob[4].cm := 204;
   		IF xZon^.cx.lck.stat = SINT_TO_USINT(xAla^.cf.typ) THEN
		   	xR^.o.ob[0].FgC := 3;
    			xR^.o.ob[0].BgC := 1;
			END_IF;

	 150: //TIMER
			xTim	:= xDev;
//			xR^.o.ob[6] 		:= _NhBrwObj.rgbwa;	//_NhBrwObj.dlgl;										// obrazok vseobecneho listu
//_NhBrwObj.dlgl
//			xR^.o.ob[7] 		:= _NhBrwObj.tim_1;										// obrazok vseobecneho listu
	 		x4o    			:= ADR(xR^.o.ob[7]);
			IF xTim^.cf.typ < 2 THEN

(*

						 	x4o    			:= ADR(xR^.o.ob[7]);
							xR^.o.ob[1].cm := 128;									// click na hlavnu ikonu = oznacovanie
							x4o^.wh			:= 107;
							x4o^.obj			:= 1;
   	 					x4o^.wxy[1]    := 52;
    						x4o^.wxy[2]    := 42;
							x4o^.obr[1]		:= 44;
							x4o^.obr[2]		:= 38;
							x4o^.ok[1] 		:= xU^.o[1].wh = xR^.h.cf.n;
							x4o^.ok[2] 		:= xRol^.me.cpy;

				_Nh_Shw_107_ROM(off:=1, o:=7);			// vypne zobrazenie nad hl.obrazkom
*)       END_IF;
				_Nh_Shw_107_ROM(off:=1, o:=8);
				blk	:= 5;

      ELSE
         IF xR^.h.cf.c > 0 THEN
				IF aCfg[xR^.h.cf.c].fbr = 15 THEN											// PODLA FORMULARA BROWSU
              	// DOR
						blk	:= 5;
						IF xA^.admin  THEN
						ELSE
                     xR^.o.ob[6].wh :=  0;                        // u WSB vypne predvolby
                     xR^.o.ob[2].cm :=  0;                        // u WSB vypne predvolby
						END_IF;
              ELSIF aCfg[xR^.h.cf.c].fbr = 20 THEN
					  // LUX,TER,TEH,TEK, 41=CO2
						_Nh_Shw_B20_ROW();
   					blk	:= 6;
	           ELSIF 	aCfg[xR^.h.cf.c].fbr = 43 							// SVD,SVA,RGB,ZAS,32=SIR,49=VVO
	           		OR aCfg[xR^.h.cf.c].fbr =  5 THEN					// SCN,ACT,DLS,DLG,DLM
		            _Nh_Frm_STA_OU(obj:=2, o:=8);
						IF aCfg[xR^.h.cf.c].analog THEN
		         	   _Nh_Frm_Row_O13(off:=xR^.h.pir ,ob:=5);
						ELSIF xM^.set THEN
//							blk 					:= 5;
							xR^.o.ob[5].wh    := 0;
						ELSE
							xR^.o.ob[5].wh    := 0;
						END_IF;
            ELSE
            ;
            END_IF;
      	END_IF;
	END_CASE;

	IF xM^.set AND new AND blk > 0 THEN
		_Nh_DEF_VAR(wh:=20, o:=blk, x:=ADR(xDev^.cf.blk));

//		xR^.o.ob[blk].x     := 125;
		xR^.o.ob[blk].w     := 48;
		xR^.o.ob[blk].h     := 48;
		xR^.o.ob[blk].FgC   := 4;
		xR^.o.ob[blk].BgC   := 2;
		xR^.o.ob[blk].fn    := 0;

	END_IF;

	{$ END_IF }
END_FUNCTION

(* ---- _Nh_UTIL.st ---- *)
FUNCTION _Nh_LoadNewPackage : BOOL
	VAR
   	rqNewProg   : BOOL;
		jak         : BOOL;
   	newPckgName : STRING := 'WWW/UPLOAD/NEW_PACK.TTR'; //http://192.168.33.200/UPLOAD/200%20v2-0-00000-00000%20PROG_PCKG%202025-09-12_16-35-57.TTR
	END_VAR
	 IF rqNewProg THEN
		jak := LoadNewPackage2( rq := rqNewProg, pckg := newPckgName);
   	rqNewProg := 0;
	END_IF;
END_FUNCTION

FUNCTION _Nh_Service_ResetToNewCfg : BOOL

END_FUNCTION

FUNCTION _Nh_Service_LoadLastOkRBx : BOOL

END_FUNCTION

 (*
 PROGRAM ExampleLoadPackage

 VAR

   rqNewProg   : BOOL;

   jak         : BOOL;

   newPckgName : STRING := 'WWW/UPLOAD/NEW_PACK.TTR';

 END_VAR

 IF rqNewProg THEN

   jak := LoadNewPackage2( rq := rqNewProg, pckg := newPckgName);

   rqNewProg := 0;

 END_IF;

END_PROGRAM
*)
